FUNCTION_BLOCK FB_MaintenanceAlarmProfile IMPLEMENTS I_AlarmProfile
VAR_INPUT
END_VAR
VAR_OUTPUT
END_VAR
VAR
END_VAR

METHOD GetName  : STRING
VAR_INPUT
END_VAR

GetName := 'MAINTENANCE';
END_METHOD

METHOD GetVoteAlert : INT
VAR_INPUT
END_VAR

GetVoteAlert     := 2;   // need 2 sensors before alerting
END_METHOD

METHOD GetVoteEmergency : INT
VAR_INPUT
END_VAR

GetVoteEmergency := 4;   // higher bar during planned maintenance
END_METHOD

METHOD GetVoteWarning  : INT
VAR_INPUT
END_VAR

GetVoteWarning   := 3;   // relaxed — maintenance activity expected
END_METHOD

END_FUNCTION_BLOCK

(* stored: Version 1.1.0.1, ProductVersion 3.1.4024.16
   POU FB_MaintenanceAlarmProfile: Id {8ee66c1d-e511-440d-b602-0ab983401346}, SpecialFunc None
   Method GetName: Id {83a671fc-ce0c-4163-8157-c91d45575af6}
   Method GetVoteAlert: Id {f73f2000-7413-46f2-8356-577687133c19}
   Method GetVoteEmergency: Id {543a43be-571e-4bb3-8b74-1de401565e28}
   Method GetVoteWarning: Id {07377599-dee2-482d-84bd-b35d76c935a6} *)
